// TIA Portal V18 export
TYPE "LGasp_typeHMI_safetydevice"
// stored: IsFailsafeCompliant false
   STRUCT
      tipo : DInt;   // 1=SBF 2=SBAA 3=BF1 4=BFM 5=TCR
      conn : WString[12];   // [XCnnn]
      intervenuto : Bool;   // attuatore intervenuto
      ninterventi : DInt;   // Numero di commutazioni
      dadefinire1 : DInt;
      dadefinire2 : DInt;
      dadefinire3 : DInt;
   END_STRUCT;
END_TYPE
